PROGRAM PRG_SMARACT
VAR
    (*
    {attribute 'TcLinkToOSO' := '
        .stDS402Drive.nModeOfOperationNC	:=<0,8,0>TINC^NC-Task 1^Axes^M9_DREAM_DGPD_MMT_Y^Drive^Outputs^Out^nCtrl5;
        .stDS402Drive.nDS402DriveControlNC := <0,8,0>TINC^NC-Task 1^Axes^M9_DREAM_DGPD_MMT_Y^Drive^Outputs^Out^nCtrl1;
        .stDS402Drive.nDS402DriveControlNC := <8,8,0>TINC^NC-Task 1^Axes^M9_DREAM_DGPD_MMT_Y^Drive^Outputs^Out^nCtrl2
    '}
    {attribute 'TcLinkTo' := '
        .stDS402Drive.nSlaveAddr:=TIID^Device 1 (EtherCAT)^B940_009_R19_DRL_02_E0_EK1200^R19_DRL_02_E4_EK1122^TMO-DREAM-SMARACT-03^InfoData^AdsAddr^port;
        .stDS402Drive.stDS402DriveStatus:=TIID^Device 1 (EtherCAT)^B940_009_R19_DRL_02_E0_EK1200^R19_DRL_02_E4_EK1122^TMO-DREAM-SMARACT-03^DREAM:DGPD:MMT:Y^mode/status/pos/fError TxPDO^Status Word;
        .stDS402Drive.nFollowingError:=;TIID^Device 1 (EtherCAT)^B940_009_R19_DRL_02_E0_EK1200^R19_DRL_02_E4_EK1122^TMO-DREAM-SMARACT-03^DREAM:DGPD:MMT:Y^mode/status/pos/fError TxPDO^Following Error Actual Value;
        .stDS402Drive.nModeOfOperation:=TIID^Device 1 (EtherCAT)^B940_009_R19_DRL_02_E0_EK1200^R19_DRL_02_E4_EK1122^TMO-DREAM-SMARACT-03^DREAM:DGPD:MMT:Y^ctl/mode/pos RxPDO^Modes of Operation;
        .stDS402Drive.nModeOfOperationDisplay:=TIID^Device 1 (EtherCAT)^B940_009_R19_DRL_02_E0_EK1200^R19_DRL_02_E4_EK1122^TMO-DREAM-SMARACT-03^DREAM:DGPD:MMT:Y^mode/status/pos/fError TxPDO^Modes of Operation Display;
        .stDS402Drive.nDS402DriveControl:=TIID^Device 1 (EtherCAT)^B940_009_R19_DRL_02_E0_EK1200^R19_DRL_02_E4_EK1122^TMO-DREAM-SMARACT-03^DREAM:DGPD:MMT:Y^ctl/mode/pos RxPDO^Control Word
    '}
    fb_DGPD_Y : FB_MotionStageMCS2CSP ( stPiezoStage:=Main.M9, eModule:=E_Module.CHAN1 );
         {attribute 'TcLinkToOSO' := '
        .stDS402Drive.nModeOfOperationNC	:=<0,8,0>TINC^NC-Task 1^Axes^M10_DREAM_DGPD_MMT_X^Drive^Outputs^Out^nCtrl5;
        .stDS402Drive.nDS402DriveControlNC := <0,8,0>TINC^NC-Task 1^Axes^M10_DREAM_DGPD_MMT_X^Drive^Outputs^Out^nCtrl1;
        .stDS402Drive.nDS402DriveControlNC := <8,8,0>TINC^NC-Task 1^Axes^M10_DREAM_DGPD_MMT_X^Drive^Outputs^Out^nCtrl2
    '}
    {attribute 'TcLinkTo' := '
        .stDS402Drive.nSlaveAddr:=TIID^Device 1 (EtherCAT)^B940_009_R19_DRL_02_E0_EK1200^R19_DRL_02_E4_EK1122^TMO-DREAM-SMARACT-03^InfoData^AdsAddr^port;
        .stDS402Drive.stDS402DriveStatus:=TIID^Device 1 (EtherCAT)^B940_009_R19_DRL_02_E0_EK1200^R19_DRL_02_E4_EK1122^TMO-DREAM-SMARACT-03^DREAM:DGPD:MMT:X^mode/status/pos/fError TxPDO^Status Word;
        .stDS402Drive.nFollowingError:=TIID^Device 1 (EtherCAT)^B940_009_R19_DRL_02_E0_EK1200^R19_DRL_02_E4_EK1122^TMO-DREAM-SMARACT-03^DREAM:DGPD:MMT:X^mode/status/pos/fError TxPDO^Following Error Actual Value;
        .stDS402Drive.nModeOfOperation:=TIID^Device 1 (EtherCAT)^B940_009_R19_DRL_02_E0_EK1200^R19_DRL_02_E4_EK1122^TMO-DREAM-SMARACT-03^DREAM:DGPD:MMT:X^ctl/mode/pos RxPDO^Modes of Operation;
        .stDS402Drive.nModeOfOperationDisplay:=TIID^Device 1 (EtherCAT)^B940_009_R19_DRL_02_E0_EK1200^R19_DRL_02_E4_EK1122^TMO-DREAM-SMARACT-03^DREAM:DGPD:MMT:X^mode/status/pos/fError TxPDO^Modes of Operation Display;
        .stDS402Drive.nDS402DriveControl:=TIID^Device 1 (EtherCAT)^B940_009_R19_DRL_02_E0_EK1200^R19_DRL_02_E4_EK1122^TMO-DREAM-SMARACT-03^DREAM:DGPD:MMT:X^ctl/mode/pos RxPDO^Control Word
    '}
    fb_DGPD_X : FB_MotionStageMCS2CSP ( stPiezoStage:=Main.M10, eModule:=E_Module.CHAN2 );
       {attribute 'TcLinkToOSO' := '
        .stDS402Drive.nModeOfOperationNC	:=<0,8,0>TINC^NC-Task 1^Axes^M11_DREAM_DGPD_MMT_RET^Drive^Outputs^Out^nCtrl5;
        .stDS402Drive.nDS402DriveControlNC := <0,8,0>TINC^NC-Task 1^Axes^M11_DREAM_DGPD_MMT_RET^Drive^Outputs^Out^nCtrl1;
        .stDS402Drive.nDS402DriveControlNC := <8,8,0>TINC^NC-Task 1^Axes^M11_DREAM_DGPD_MMT_RET^Drive^Outputs^Out^nCtrl2
    '}
    {attribute 'TcLinkTo' := '
        .stDS402Drive.nSlaveAddr:=TIID^Device 1 (EtherCAT)^B940_009_R19_DRL_02_E0_EK1200^R19_DRL_02_E4_EK1122^TMO-DREAM-SMARACT-03^InfoData^AdsAddr^port;
        .stDS402Drive.stDS402DriveStatus:=TIID^Device 1 (EtherCAT)^B940_009_R19_DRL_02_E0_EK1200^R19_DRL_02_E4_EK1122^TMO-DREAM-SMARACT-03^DREAM:DGPD:MMT:RET^mode/status/pos/fError TxPDO^Status Word;
        .stDS402Drive.nFollowingError:=TIID^Device 1 (EtherCAT)^B940_009_R19_DRL_02_E0_EK1200^R19_DRL_02_E4_EK1122^TMO-DREAM-SMARACT-03^DREAM:DGPD:MMT:RET^mode/status/pos/fError TxPDO^Following Error Actual Value;
        .stDS402Drive.nModeOfOperation:=TIID^Device 1 (EtherCAT)^B940_009_R19_DRL_02_E0_EK1200^R19_DRL_02_E4_EK1122^TMO-DREAM-SMARACT-03^DREAM:DGPD:MMT:RET^ctl/mode/pos RxPDO^Modes of Operation;
        .stDS402Drive.nModeOfOperationDisplay:=TIID^Device 1 (EtherCAT)^B940_009_R19_DRL_02_E0_EK1200^R19_DRL_02_E4_EK1122^TMO-DREAM-SMARACT-03^DREAM:DGPD:MMT:RET^mode/status/pos/fError TxPDO^Modes of Operation Display;
        .stDS402Drive.nDS402DriveControl:=TIID^Device 1 (EtherCAT)^B940_009_R19_DRL_02_E0_EK1200^R19_DRL_02_E4_EK1122^TMO-DREAM-SMARACT-03^DREAM:DGPD:MMT:RET^ctl/mode/pos RxPDO^Control Word
    '}
    fb_DGPD_RET : FB_MotionStageMCS2CSP ( stPiezoStage:=Main.M11, eModule:=E_Module.CHAN3 );

    stDGPD_RET: ARRAY[1..GeneralConstants.MAX_STATES] OF ST_PositionState;

    {attribute 'pytmc' := '
          pv: DGPD:RET:STATES:SET
          io: io
    '}
     stDGPD_RET_Set: ENUM_AxisStates;
        {attribute 'pytmc' := '
          pv: DGPD:RET:STATES:GET
          io: i
        '}
    stDGPD_RET_Get: ENUM_AxisStates;

    fbDGPD_RET_PMPStates: FB_PositionStatePMPS1D;
    *)
END_VAR

(*
fbDGPD_RET_PMPStates(
    stMotionStage:=Main.M11,
    astPositionState:=stDGPD_RET,
    eEnumSet:=stDGPD_RET_Set,
    eEnumGet:=stDGPD_RET_Get,
    sDeviceName := 'DREAM:DGPD:MMT:RET',
    sTransitionKey := 'DREAM:DGPD:MMT:RET-TRANSITION',
    fbFFHWO:=GVL_PMPS.fbFastFaultOutput1,
    fbArbiter:=GVL_PMPS.fbArbiter1,
    bEnableMotion:=TRUE,
    bEnableBeamParams:=TRUE,
    bEnablePositionLimits:=TRUE,
    bReadDBNow:=TRUE,
);

fb_DGPD_RET();
fb_DGPD_X();
fb_DGPD_Y();
*)

END_PROGRAM

(* stored: Version 1.1.0.1
   POU PRG_SMARACT: Id {8c8a4af2-8a7c-4f25-948f-bede85609ff3}, SpecialFunc None *)
